Universal Robots URScript: generic_movel.urscript

def go_to_home():
	movel(p[{}, {}, {}, {}, {}, {}])
end
